# B&R Automation Studio project CombinedLinenCleanA6 (part 4)

#### usb_pmem.ab
```automation-basic
;--------------------------------------------------------------
;Copy BagData, C and D data to and from USB Mass Storage device
;--------------------------------------------------------------

;----------------------------------------------------
;Version 1.00 05/08/2006 D.J. First Issue
;Version 2.00 24/06/2009 D.J. Added D32 & VC_Posn
;Version 3.00 03/11/2010 D.J. Changed VC to RB (Robo)
;----------------------------------------------------

;Notes:-
;Add a mass storage device to the PLC CPU
;In CPU Properties select File Device
;Add a new device and set the Device Name to "USBStick"
;set the path of the USB device eg. "IF3.ST1" for a CP340

PROGRAM _INIT

bOK 			= FALSE
STEP 			= 1
byErrorLevel 	= 0
CurrentFile 	= 0

END_PROGRAM

PROGRAM _CYCLIC

;Error Step
IF STEP = 0 THEN
	bOK = FALSE
ENDIF

;Check if the file exists
IF STEP = 1 THEN

	FOpen.enable    = TRUE
    FOpen.pDevice   = "USBStick"
    IF CurrentFile = 0 THEN
    	FOpen.pFile     = "PLC_BagData.dat"
    ELSE IF CurrentFile = 1 THEN
    	FOpen.pFile     = "PLC_C.dat"
    ELSE IF CurrentFile = 2 THEN
    	FOpen.pFile     = "PLC_D.dat"
	ELSE IF CurrentFile = 3 THEN
    	FOpen.pFile     = "PLC_D32.dat"
	ELSE IF CurrentFile = 4 THEN
    	FOpen.pFile     = "PLC_RBPosn.dat"
    ENDIF
    FOpen.mode      = 2 ;Read and write access

    FOpen FUB FileOpen()

    dwIdent = FOpen.ident
    wStatus = FOpen.status

    ;Status - 20708 = File doesn't exist
    IF (wStatus = 20708) THEN
    	STEP = 2 ;If the file not found then create the file
    ELSE
    	IF (wStatus = 0) THEN
        	STEP = 4 ;If the file exists then copy back to PLC
    	ELSE
        	IF (wStatus <> 65535) THEN
            	byErrorLevel = 1
                STEP = 0
				IF (wStatus = 20799) THEN
                	wError = FileIoGetSysError()
           		ENDIF
            ENDIF
    	ENDIF
    ENDIF

ENDIF

;Create the file
IF STEP = 2 THEN

	FCreate.enable  = TRUE
    FCreate.pDevice = "USBStick"
    IF CurrentFile = 0 THEN
    	FCreate.pFile     = "PLC_BagData.dat"
    ELSE IF CurrentFile = 1 THEN
    	FCreate.pFile     = "PLC_C.dat"
    ELSE IF CurrentFile = 2 THEN
    	FCreate.pFile     = "PLC_D.dat"
    ELSE IF CurrentFile = 3 THEN
    	FCreate.pFile     = "PLC_D32.dat"
	ELSE IF CurrentFile = 4 THEN
    	FCreate.pFile     = "PLC_RBPosn.dat"
    ENDIF
    FCreate FUB FileCreate()

    dwIdent = FCreate.ident
    wStatus = FCreate.status

    IF (wStatus = 0) THEN
    	STEP = 3
    ELSE
    	IF (wStatus <> 65535) THEN
        	byErrorLevel = 4
            STEP = 5 ;Close
			IF (wStatus = 20799) THEN
            	wError = FileIoGetSysError() ;General System Error - get more info
        	ENDIF
    	ENDIF
    ENDIF
ENDIF

;Write data to the file
IF STEP = 3 THEN

    FWrite.enable   = TRUE
    FWrite.ident    = dwIdent
    FWrite.offset   = 0
    IF CurrentFile = 0 THEN
    	FWrite.pSrc     = pBag
    	FWrite.len      = sizeof(Bag)
    ELSE IF CurrentFile = 1 THEN
    	FWrite.pSrc     = pC
    	FWrite.len      = sizeof(C)
    ELSE IF CurrentFile = 2 THEN
    	FWrite.pSrc     = pD
    	FWrite.len      = sizeof(D)
	ELSE IF CurrentFile = 3 THEN
    	FWrite.pSrc     = pD32
    	FWrite.len      = sizeof(D32)
	ELSE IF CurrentFile = 4 THEN
    	FWrite.pSrc     = pRB_Posn
    	FWrite.len      = sizeof(RB_Posn)
    ENDIF

    FWrite FUB FileWrite()

    wStatus = FWrite.status

    ;Status
    IF (wStatus = 0) THEN
    	STEP = 5 ;Close
    ELSE
       	IF (wStatus <> 65535) THEN
        	byErrorLevel = 3
    		STEP = 0

          	IF (wStatus = 20799) THEN
            	wError = FileIoGetSysError() ;General System Error - get more info
        	ENDIF
     	ENDIF
  	ENDIF
ENDIF

;Read file
IF STEP = 4 THEN

    FRead.enable    = TRUE
    FRead.ident     = dwIdent
    FRead.offset    = 0

	IF CurrentFile = 0 THEN
    	FRead.pDest     = pBag
    	FRead.len      = sizeof(Bag)
    ELSE IF CurrentFile = 1 THEN
    	FRead.pDest     = pC
    	FRead.len      = sizeof(C)
    ELSE IF CurrentFile = 2 THEN
    	FRead.pDest     = pD
    	FRead.len      = sizeof(D)
    ELSE IF CurrentFile = 3 THEN
    	FRead.pDest     = pD32
    	FRead.len      	= sizeof(D32)
	ELSE IF CurrentFile = 4 THEN
    	FRead.pDest     = pRB_Posn
    	FRead.len      	= sizeof(RB_Posn)
	ENDIF

    FRead FUB FileRead()

    wStatus = FRead.status

	;Status
    IF (wStatus = 0) THEN
    	STEP = 5
    ELSE
        IF (wStatus <> 65535) THEN
            byErrorLevel = 4
            STEP = 0
            IF (wStatus = 20799) THEN
            	wError = FileIoGetSysError() ;General System Error - get more info
            ENDIF
        ENDIF
    ENDIF
ENDIF

;Close the file
IF STEP = 5 THEN

	FClose.enable   = TRUE
	FClose.ident    = dwIdent

	FClose FUB FileClose()

	wStatus = FClose.status

	;Status
	IF (wStatus = 0) THEN
		STEP = 7
	ELSE
        IF (wStatus <> 65535) THEN
            byErrorLevel = 5
            STEP = 0

            IF (wStatus = 20799) THEN
            	wError = FileIoGetSysError() ;General System Error - get more info
            ENDIF
        ENDIF
	ENDIF
ENDIF

;Operation Complete - try next file if required
IF STEP = 7 THEN
	IF CurrentFile < 4 THEN
		CurrentFile = CurrentFile + 1
		STEP = 1
	ENDIF
ENDIF

;Set this step manually to test this routine
IF (STEP = 8) THEN
	CurrentFile = 0
	STEP		= 1
ENDIF
END_PROGRAM
```

- Program Logical/Sequences/200ms/zzAlarms (IEC, version 4.00.0) (no source held here)

### zzstn_q.var
```iecst
VAR
	n : UINT;
	ValidWeight : BOOL;
	SP1Reached : BOOL;
	SP2Reached : BOOL;
	SP3Reached : BOOL;
	TestWeight : UINT;
	StnIntoQ : BOOL;
	StnsInQ : BOOL;
	PurgeStation : BOOL;
	StnsToPurge : BOOL;
	ManualRelease : BOOL;
	TestStation : UINT;
	z : UINT;
	Calibration : BOOL;
END_VAR
```

### Program Logical/Sequences/200ms/zzTime

#### zztime.var
```iecst
VAR RETAIN
	MiliSeconds	:UINT;
	Seconds	:UINT;
END_VAR

VAR
	TEST	:BOOL;
	TimeLast	:TIME;
	TimeNow	:TIME;
	TimeDiff	:TIME;
	SysRunning	:BOOL;
	ActionPLS	:BOOL;
	NoActionET	:TIME;
	NoAction	:BOOL;
	NoActionPLS	:BOOL;
	PLCFirstScan	:BOOL;
	Seq	:UINT;
	Minutes	:INT;
	Hours	:UINT;
	SysIdleMinutes	:UINT;
	SystemAction	:BOOL;
END_VAR
```

#### zztime.ab
```automation-basic
;-------------------
;System Running Time
;-------------------

;-----------------------------------------
;Revision 1.00 12/10/2005 D.J. First Issue
;-----------------------------------------

;Detection of system running - once the detection sequence has remained idle for a given
;period the clock is stopped and the idle time (minutes) is given back. If the idle time
;is 5 minutes and the system stopped at 12:01 then when the time is given back the time will
;read 12:-04 as the time is only taken from the minutes and no the hours count.

PROGRAM _INIT

PLCFirstScan = TRUE

END_PROGRAM

PROGRAM _CYCLIC

;Only use one sequence for system running. Norrmally Offgoing or a loop use the Discharger
D[905]	;Monitor

SystemAction = FALSE
IF D[915] <> Seq THEN
	SystemAction 	= TRUE
	Seq 			= D[915]
ENDIF

R_TRIG(SystemAction,ActionPLS)

TimeNow = clock_ms()

;System Start / Stop Running
IF ActionPLS THEN
	SysRunning 	= TRUE
ENDIF

SysIdleMinutes = 5

TON_10ms(NOT SystemAction,(SysIdleMinutes * 6000),NoAction,NoActionET)

;Read from Graphics
;Seconds = D[310]
Minutes = INT(D[311]) ;Can go minus
Hours	= D[312]

R_TRIG(NoAction,NoActionPLS)

;System has stopped give back the running timer time
IF NoActionPLS THEN
	Minutes 	= Minutes - SysIdleMinutes
	SysRunning 	= FALSE
ENDIF

IF TEST THEN
	Minutes 	= Minutes - 10
	TEST 		= FALSE
ENDIF

IF SysRunning THEN
	TimeDiff	= DiffT(TimeNow,TimeLast)
	MiliSeconds = MiliSeconds + UINT(TimeDiff)
ENDIF

TimeLast = TimeNow

;Count Seconds Running
IF MiliSeconds >= 1000 THEN
	Seconds 	= Seconds + 1
	MiliSeconds = MiliSeconds - 1000 ;Keep and remaing ms to be added next time
ENDIF

IF Seconds >= 60 THEN
	Minutes 	= Minutes + 1
	Seconds 	= Seconds - 60
ENDIF

IF Minutes >= 60 THEN
	Hours 		= Hours + 1
	Minutes	 	= Minutes - 60
ENDIF

;Count Each 1000 hours
IF Hours >= 1000 THEN
	D[313] 		= D[313] + 1
	Hours 		= Hours - 1000
ENDIF

;Store to Graphics
;D[310] = Seconds - don't display seconds as causes TCP/IP driver to send data to Graphics
D[311] = UINT(Minutes)
D[312] = Hours
D[313] = D[313] ;Hours * 1000

END_PROGRAM
```

### zzweigh.typ
```iecst
(********************************************************************
 * COPYRIGHT -- HP
 ********************************************************************
 * Package: NewPackage
 * File: zzweigh.typ
 * Author: treamsbottom
 * Created: April 10, 2014
 ********************************************************************
 * Data types of package NewPackage
 ********************************************************************)

TYPE
	enum_Calib :
		(
		Calib_Low,
		Calib_High
		);
END_TYPE
```

- Data object Logical/Sequences/Robo_Drive_Control/Param_0_25kwStar1 (Simple, version 4.00.0) (no source held here)

- Data object Logical/Sequences/Robo_Drive_Control/Param_2_2kwStar (Simple, version 4.00.0) (no source held here)

- Data object Logical/Sequences/Robo_Drive_Control/ParaTest (Simple) (no source held here)

- Program Logical/Sequences/TB/12_belt2 (IEC) (no source held here)

### zcusfifo.var
```iecst
VAR RETAIN
	OngoingCus	:UINT;
	EditCus	:UINT;
	n	:UINT;
	x	:UINT;
END_VAR
```

### Program Logical/Sequences/zzalarms (IEC, version 2.00.0)

#### zzalarms.var
```iecst
VAR RETAIN
	I_CancelAlarm	:BOOL;
END_VAR

VAR
	BuildD220	:UINT;
	AlmNumber	:UINT;
	n	:UINT;
	AlarmCount	:UINT;
	CancelBeacon	:BOOL;
	I_MotorOverload	:BOOL;
	UnloadingAlarm	:BOOL;
	I_InverterFault	:BOOL;
	BeaconInList	:BOOL;
END_VAR
```

#### zzalarmsCyclic.ab
```automation-basic
PROGRAM _CYCLIC
	(* cyclic program *)

;-----------------------------------------------
;Alarm Messages with Screen position and history
;-----------------------------------------------

;------------------------------------------------
;Version 1.00 - 08/12/2005 First Issue D.J.
;Vesrion 2.00 - 17/10/2006 Added Alarm.Extra D.J.
;------------------------------------------------

;Note - Sequence must set the following
;Alarm[x].on
;Alarm[x].Bag - for the bag position where the alarm will appear
;Alarm[x].Name - for the message that will be displayed use constants strating "alm"
;Alarn[x].Extra - Extra data for Graphics to use ie. Line number with fault on offgoing storage

I_CancelAlarm 	= FALSE ;X[4].X16
I_EStop 		= Std.EStop
I_MotorOverload = Std.MotorOverload
I_InverterFault = FALSE ;(X[3].X03 OR X[3].X04 OR X[3].X05 OR X[3].X06)

;--------------
;Alarm Messages
;--------------

IF I_EStop THEN
	Alarm[100].On	= TRUE
	Alarm[100].Bag 	= 0
	Alarm[100].Name	= almEmergencyStop
ELSE IF I_MotorOverload THEN
	Alarm[100].On	= TRUE
	Alarm[100].Bag 	= 0
	Alarm[100].Name	= almMotorOverload
ELSE IF I_InverterFault THEN
	Alarm[100].On	= TRUE
	Alarm[100].Bag 	= 0
	Alarm[100].Name	= almInverterFault
ELSE
	Alarm[100].On	= FALSE
	Alarm[100].Bag 	= 0
	Alarm[100].Name	= almNoAlarm
ENDIF

;Shuffle the Alarms List

AlarmCount 		= 0
BeaconInList 	= FALSE

LOOP n = 1 TO 10 DO

	;If Alarm not on anymore the clear from the list
	AlmNumber = D[200 + n]
	IF NOT Alarm[AlmNumber].On THEN
		D[200 + n] = 0
		D[210 + n] = 0
	ENDIF

	;Shuffle the list down
	IF (D[200 + n] = 0) AND (D[201 + n] > 0) AND (n <> 10) THEN
		D[200 + n] = D[201 + n]
		D[210 + n] = D[211 + n]
		D[201 + n] = 0
		D[211 + n] = 0
	ENDIF

	;Set InList for any alarm in the list
	Alarm[D[200 + n]].InList = TRUE

	;Calculate total alarms in the list
	IF D[200 + n] > 0 THEN
		AlarmCount = AlarmCount + 1
	ENDIF

	;Is the alarm beacon required?
	IF Alarm[AlmNumber].On AND Alarm[AlmNumber].Beacon THEN
		BeaconInList = TRUE
	ENDIF

ENDLOOP

;Cancel the alarm beacon
IF I_CancelAlarm THEN
	CancelBeacon = TRUE
ENDIF

;Cancel the CancelAlarm beacon if no alarm in the list requires the beacon
IF NOT BeaconInList THEN
	CancelBeacon = FALSE
ENDIF

;Look at each sequence alarm and if not in list then add to list if space
LOOP n = 1 TO 109 DO

	;If alarm active and a code has been given and not in the list and history is clear then add
	IF ((AlarmCount < 10) AND Alarm[n].On AND NOT Alarm[n].InList AND ((D[221] = 0) OR (n > 100))) THEN

		;If name not set then set to general
		IF (Alarm[n].Name = 0) THEN
			Alarm[n].Name = almGeneralSequence
		ENDIF

		D[210] 			= n
		BuildD220		= LSL(Alarm[n].Extra,8)
		BuildD220 		= BuildD220 + Alarm[n].Name
		D[220] 			= BuildD220

		;New alarm found requiring the beacon
		IF Alarm[n].Beacon THEN
			CancelBeacon = FALSE
		ENDIF

		;Store to History - if not Unloading Alarm
		IF (n <= 100) THEN
			D[221] 			= n				;Alarm Number (Seq)
			D[222]			= Alarm[n].Name	;Alarm Name / Message
			D[223] 			= D[223] + 1	;Alarm ID
			D[224]			= Alarm[n].Extra;Alarm Extra Data
			IF D[223] > 32000 THEN
				D[223] = 1
			ENDIF
		ENDIF

		;Inc Total Alarms
		AlarmCount = AlarmCount + 1

	ENDIF

	;Cancel All InList's - will be checked on the next scan
	Alarm[n].InList = FALSE

ENDLOOP

;Show Alarm position on the screen
IF D[201] > 0 THEN
	D[0] = Alarm[D[201]].Bag
ELSE
	D[0] = 0
ENDIF

UnloadingAlarm = Alarm[101].On OR Alarm[102].On OR Alarm[103].On OR Alarm[104].On

;Alarm Output - Unloading Alarm cannot be cancelled
Y[3].Y16 = ((BeaconInList AND NOT CancelBeacon) OR UnloadingAlarm)
;Y[4].Y15 = CancelAlarm
END_PROGRAM
```

### Program Logical/Sequences/zzbagsfl

#### zzbagsfl.var
```iecst
VAR RETAIN
	CurrentBag	:UINT;
	CurrentLine	:UINT;
	LineSp	:UINT;
END_VAR

VAR
	NextBag	:UINT;
END_VAR
```

#### zzbagsflCyclic.ab
```automation-basic
PROGRAM _CYCLIC
	(* cyclic program *)

;-----------------------------------------------------------
;Revision 1.00 19/12/2005 D.J. First Issue - Using BAG array
;-----------------------------------------------------------

Std.BagsWithDestinations 	= FALSE
Std.CustomerFound	 		= FALSE

IF (Bag[75].Cat>0)AND (Bag[5].Cat=0)THEN
		Bag[5] = Bag[75]
		Bag[75] = Bag[0]
ENDIF
IF (Bag[70].Cat>0)AND (Bag[20].Cat=0)THEN
		Bag[20] = Bag[70]
		Bag[70] = Bag[0]
ENDIF

LOOP CurrentLine = 1 to Std.MaxLinesBuffers DO

	LineSp = 0

	LOOP CurrentBag = Line[CurrentLine].FirstBag  TO Line[CurrentLine].LastBag DO

		EXITIF Line[CurrentLine].FirstBag = 0

		NextBag = (CurrentBag + 1)

		IF ((CurrentBag < Line[CurrentLine].LastBag) AND ((Bag[CurrentBag].Cat = 0) AND (Bag[NextBag].Cat > 0))) THEN

			;Copy Next Bag to Current
			Bag[CurrentBag]	= Bag[NextBag]
			Bag[NextBag] 	= Bag[0]

		ENDIF

		IF ((Bag[CurrentBag].Dst > 0) AND (CurrentLine <= Std.MaxLines)) THEN
			Std.BagsWithDestinations = TRUE
		ENDIF

		;Add the line spaces up
		IF Bag[CurrentBag].Cat = 0 THEN
			LineSp = (LineSp + 1)
		ENDIF

		;For Customer FIFO table
		;-----------------------
		;Customer at front of FIFO in Storage
		IF ((Bag[CurrentBag].Cus = D[401]) AND (D[401] > 0) AND (CurrentLine <= Std.MaxLines)) THEN
			Std.CustomerFound	 	= TRUE
		ENDIF

	ENDLOOP
	;Save the number of spaces on the current line
	Line[CurrentLine].Space = LineSp

ENDLOOP

Line[4].Space = (Line[4].Space + Line[10].Space)
Line[1].Space = (Line[1].Space + Line[11].Space)

END_PROGRAM
```

### Program Logical/Sequences/zzbitcal

#### zzbitcalCyclic.ab
```automation-basic
PROGRAM _CYCLIC
	(* cyclic program *)

	;-----------------------------------------------------------
	;Revision 1.00 19/12/2005 D.J. First Issue - Using BAG array
	;-----------------------------------------------------------

	;Find the Space on each Storage line including the Ongoing and Offgoing Bags In Transit

	;See Init Routine - Change settings for bags in transit bag numbers

	;Clear local calculation
	LOOP n = 1 TO Std.MaxLinesBuffers DO
		SpaceBIT[n] = 0
	ENDLOOP

	;Ensure the destination is less than the Array size of SpaceBIT	(normally 100)
	LOOP n = 1 TO TotalTransitBags DO
		Destination = Bag[BITDest[n]].Dst
		IF (Destination > 0) AND (Destination < 100) THEN
			SpaceBIT[Destination] = SpaceBIT[Destination] + 1
		ENDIF
	ENDLOOP

	;Once all calculated then update the global line space
	LOOP n = 1 TO Std.MaxLinesBuffers DO
		Spaces = (INT(Line[n].Space) - INT(SpaceBIT[n]))
		IF Spaces > 0 THEN
			Line[n].SpaceBIT = UINT(Spaces)
		ELSE
			Line[n].SpaceBIT = 0
		ENDIF
	ENDLOOP

END_PROGRAM
```

#### zzbitcalInit.ab
```automation-basic
PROGRAM _INIT
	(* init program *)

BITBag = 1

;Transfer Belt Bags - Pair loop
LOOP n = 32 TO 59 DO
	BITDest[BITBag] = n
	BITBag = BITBag + 1
ENDLOOP

;Bags in transit
;LOOP n = 140 to 179 DO
	;BITDest[BITBag] = n
	;BITBag = BITBag + 1
;ENDLOOP

TotalTransitBags = (BITBag - 1)
END_PROGRAM
```

- Program Logical/Sequences/zzclrmem (IEC, version 2.00.0) (no source held here)

### Program Logical/Sequences/zzconst (IEC, version 1.00.0)

#### zzconstInit.ab
```automation-basic
PROGRAM _INIT
	(* init program *)

Std.AutoMaticRelease   	= TRUE	;Set to TRUE for AutoMatic Release using setpoints. FALSE for Push-Button Release
Std.StationReports  	= TRUE  ;Transfer reports to PC

Std.PairingLoop   		= FALSE
Std.CustomerFIFO		= TRUE	;Use Customer FIFO Table

Std.MaxIO				= 39	;Max PLC I/O Cards - check X and Y array size

Std.MaxCats           	= 99	;Max Categories - Should be 99 or less Max = 255
Std.MaxCust           	= 999	;Max Customers
Std.MaxDischargers    	= 2		;Total Dischargers
Std.MaxLines          	= 11	    ;Max storage lines
Std.MaxLinesBuffers   	= 18	;Storage lines + Buffers
Std.MaxWeighstations  	= 16	    ;Total Weighstations
Std.MaxStationBanks		= 1		;Total Banks of sorting Stations
Std.MaxSearch			= 2    	;Include all station banks and Loading VC's etc
Std.StationBagsStart[1]	= 201	;Bag Number of first bank of sorting stations
Std.StationBagsStart[2] = 0 	;Bag Number of second bank of sorting stations
Std.MinReleaseWeight  	= 30	;Include 10ths Norm 30

Ldg[1].StartStn 		= 1 	;Bank 1 Start station number
Ldg[1].EndStn			= 16	    ;Bank 1 End station number

Ldg[2].StartStn 		= 0 	;Bank 2 Start station number
Ldg[2].EndStn			= 0		;Bank 2 End station number

;Enter the First and Last bag for all the Storage lines including buffers
Line[1].FirstBag = 1
Line[1].LastBag  = 5

Line[2].FirstBag = 6
Line[2].LastBag  = 10

Line[3].FirstBag = 11
Line[3].LastBag  = 13

Line[4].FirstBag = 16
Line[4].LastBag  = 20

Line[5].FirstBag = 26
Line[5].LastBag  = 29

Line[6].FirstBag = 21
Line[6].LastBag  = 24

Line[7].FirstBag = 63  ;New line for cdc7
Line[7].LastBag  = 66

Line[8].FirstBag = 78  ;New line for cdc8
Line[8].LastBag  = 81

Line[9].FirstBag = 0
Line[9].LastBag  = 0

Line[10].FirstBag = 70  ;Part of line 1
Line[10].LastBag  = 72

Line[11].FirstBag = 75  ;Part of line 4
Line[11].LastBag  = 77

Line[12].FirstBag = 0
Line[12].LastBag  = 0

Line[13].FirstBag = 0
Line[13].LastBag  = 0

Line[14].FirstBag = 0
Line[14].LastBag  = 0

Line[15].FirstBag = 0
Line[15].LastBag  = 0

Line[16].FirstBag = 51
Line[16].LastBag  = 52

Line[17].FirstBag = 38
Line[17].LastBag  = 38

Line[18].FirstBag = 53    ;New line for CP16
Line[18].LastBag  = 53

Line[19].FirstBag = 0
Line[19].LastBag  = 0

Line[20].FirstBag = 0
Line[20].LastBag  = 0

Line[21].FirstBag = 227
Line[21].LastBag  = 227

Line[22].FirstBag = 229
Line[22].LastBag  = 230

Line[23].FirstBag = 0
Line[23].LastBag  = 0

Line[24].FirstBag = 0
Line[24].LastBag  = 0

Line[25].FirstBag = 0
Line[25].LastBag  = 0

Line[26].FirstBag = 0
Line[26].LastBag  = 0

Line[27].FirstBag = 0
Line[27].LastBag  = 0

Line[28].FirstBag = 0
Line[28].LastBag  = 0

Line[29].FirstBag = 0
Line[29].LastBag  = 0

Line[30].FirstBag = 0
Line[30].LastBag  = 0

Line[31].FirstBag = 0
Line[31].LastBag  = 0

Line[32].FirstBag = 0
Line[32].LastBag  = 0

Line[33].FirstBag = 0
Line[33].LastBag  = 0

Line[34].FirstBag = 0
Line[34].LastBag  = 0
END_PROGRAM
```

#### zzconstCyclic.ab
```automation-basic
PROGRAM _CYCLIC
	(* cyclic program *)
;-----------------------------------------------------
;Revision A 01/05/2001 D.J. First Issue
;-----------------------------------------------------
;Code In Init Subroutine

Std.EnableOverUnderRelease = FALSE ;X6C 	;Override KeySwitch - See Stn_Q
END_PROGRAM
```

### Program Logical/Sequences/zzforcei

#### zzforcei.var
```iecst
VAR
	n	:UINT;
	XForce	:CardInputs;
	XForceVal	:CardInputs;
END_VAR
```

#### zzforceiCyclic.ab
```automation-basic
PROGRAM _CYCLIC
(* cyclic program *)

;---------------------------
;Input forcing from Graphics
;---------------------------

;Version 1.00 14/09/2006 D.J. First Issue

n = D[303]

IF (n > Std.MaxIO) THEN
	n = 0
ENDIF

XForce.X01 		= BIT_TST(D[304],0)
XForce.X02 		= BIT_TST(D[304],1)
XForce.X03 		= BIT_TST(D[304],2)
XForce.X04 		= BIT_TST(D[304],3)
XForce.X05 		= BIT_TST(D[304],4)
XForce.X06 		= BIT_TST(D[304],5)
XForce.X07 		= BIT_TST(D[304],6)
XForce.X08 		= BIT_TST(D[304],7)
XForce.X09 		= BIT_TST(D[304],8)
XForce.X10 		= BIT_TST(D[304],9)
XForce.X11 		= BIT_TST(D[304],10)
XForce.X12 		= BIT_TST(D[304],11)
XForce.X13 		= BIT_TST(D[304],12)
XForce.X14 		= BIT_TST(D[304],13)
XForce.X15 		= BIT_TST(D[304],14)
XForce.X16 		= BIT_TST(D[304],15)

XForceVal.X01 	= BIT_TST(D[305],0)
XForceVal.X02 	= BIT_TST(D[305],1)
XForceVal.X03 	= BIT_TST(D[305],2)
XForceVal.X04 	= BIT_TST(D[305],3)
XForceVal.X05 	= BIT_TST(D[305],4)
XForceVal.X06 	= BIT_TST(D[305],5)
XForceVal.X07 	= BIT_TST(D[305],6)
XForceVal.X08 	= BIT_TST(D[305],7)
XForceVal.X09 	= BIT_TST(D[305],8)
XForceVal.X10 	= BIT_TST(D[305],9)
XForceVal.X11 	= BIT_TST(D[305],10)
XForceVal.X12 	= BIT_TST(D[305],11)
XForceVal.X13 	= BIT_TST(D[305],12)
XForceVal.X14 	= BIT_TST(D[305],13)
XForceVal.X15 	= BIT_TST(D[305],14)
XForceVal.X16 	= BIT_TST(D[305],15)

X[n].X01 = (X[n].X01 AND NOT XForce.X01) OR (XForce.X01 AND XForceVal.X01)
X[n].X02 = (X[n].X02 AND NOT XForce.X02) OR (XForce.X02 AND XForceVal.X02)
X[n].X03 = (X[n].X03 AND NOT XForce.X03) OR (XForce.X03 AND XForceVal.X03)
X[n].X04 = (X[n].X04 AND NOT XForce.X04) OR (XForce.X04 AND XForceVal.X04)
X[n].X05 = (X[n].X05 AND NOT XForce.X05) OR (XForce.X05 AND XForceVal.X05)
X[n].X06 = (X[n].X06 AND NOT XForce.X06) OR (XForce.X06 AND XForceVal.X06)
X[n].X07 = (X[n].X07 AND NOT XForce.X07) OR (XForce.X07 AND XForceVal.X07)
X[n].X08 = (X[n].X08 AND NOT XForce.X08) OR (XForce.X08 AND XForceVal.X08)
X[n].X09 = (X[n].X09 AND NOT XForce.X09) OR (XForce.X09 AND XForceVal.X09)
X[n].X10 = (X[n].X10 AND NOT XForce.X10) OR (XForce.X10 AND XForceVal.X10)
X[n].X11 = (X[n].X11 AND NOT XForce.X11) OR (XForce.X11 AND XForceVal.X11)
X[n].X12 = (X[n].X12 AND NOT XForce.X12) OR (XForce.X12 AND XForceVal.X12)
X[n].X13 = (X[n].X13 AND NOT XForce.X13) OR (XForce.X13 AND XForceVal.X13)
X[n].X14 = (X[n].X14 AND NOT XForce.X14) OR (XForce.X14 AND XForceVal.X14)
X[n].X15 = (X[n].X15 AND NOT XForce.X15) OR (XForce.X15 AND XForceVal.X15)
X[n].X16 = (X[n].X16 AND NOT XForce.X16) OR (XForce.X16 AND XForceVal.X16)
END_PROGRAM
```

### Program Logical/Sequences/zzforceo

#### zzforceo.var
```iecst
VAR
	YForce	:CardOutputs;
	YForceVal	:CardOutputs;
	n	:UINT;
END_VAR
```

#### zzforceoCyclic.ab
```automation-basic
PROGRAM _CYCLIC
(* cyclic program *)

;----------------------------
;Output forcing from Graphics
;----------------------------

;Version 1.00 02/09/2006 D.J. First Issue

n = D[303]

IF (n > Std.MaxIO) THEN
	n = 0
ENDIF

YForce.Y01 		= BIT_TST(D[306],0)
YForce.Y02 		= BIT_TST(D[306],1)
YForce.Y03 		= BIT_TST(D[306],2)
YForce.Y04 		= BIT_TST(D[306],3)
YForce.Y05 		= BIT_TST(D[306],4)
YForce.Y06 		= BIT_TST(D[306],5)
YForce.Y07 		= BIT_TST(D[306],6)
YForce.Y08 		= BIT_TST(D[306],7)
YForce.Y09 		= BIT_TST(D[306],8)
YForce.Y10 		= BIT_TST(D[306],9)
YForce.Y11 		= BIT_TST(D[306],10)
YForce.Y12 		= BIT_TST(D[306],11)
YForce.Y13 		= BIT_TST(D[306],12)
YForce.Y14 		= BIT_TST(D[306],13)
YForce.Y15 		= BIT_TST(D[306],14)
YForce.Y16 		= BIT_TST(D[306],15)

YForceVal.Y01 	= BIT_TST(D[307],0)
YForceVal.Y02 	= BIT_TST(D[307],1)
YForceVal.Y03 	= BIT_TST(D[307],2)
YForceVal.Y04 	= BIT_TST(D[307],3)
YForceVal.Y05 	= BIT_TST(D[307],4)
YForceVal.Y06 	= BIT_TST(D[307],5)
YForceVal.Y07 	= BIT_TST(D[307],6)
YForceVal.Y08 	= BIT_TST(D[307],7)
YForceVal.Y09 	= BIT_TST(D[307],8)
YForceVal.Y10 	= BIT_TST(D[307],9)
YForceVal.Y11 	= BIT_TST(D[307],10)
YForceVal.Y12 	= BIT_TST(D[307],11)
YForceVal.Y13 	= BIT_TST(D[307],12)
YForceVal.Y14 	= BIT_TST(D[307],13)
YForceVal.Y15 	= BIT_TST(D[307],14)
YForceVal.Y16 	= BIT_TST(D[307],15)

Y[n].Y01 = (Y[n].Y01 AND NOT YForce.Y01) OR (YForce.Y01 AND YForceVal.Y01 AND NOT YForceDisable[n].Y01)
Y[n].Y02 = (Y[n].Y02 AND NOT YForce.Y02) OR (YForce.Y02 AND YForceVal.Y02 AND NOT YForceDisable[n].Y02)
Y[n].Y03 = (Y[n].Y03 AND NOT YForce.Y03) OR (YForce.Y03 AND YForceVal.Y03 AND NOT YForceDisable[n].Y03)
Y[n].Y04 = (Y[n].Y04 AND NOT YForce.Y04) OR (YForce.Y04 AND YForceVal.Y04 AND NOT YForceDisable[n].Y04)
Y[n].Y05 = (Y[n].Y05 AND NOT YForce.Y05) OR (YForce.Y05 AND YForceVal.Y05 AND NOT YForceDisable[n].Y05)
Y[n].Y06 = (Y[n].Y06 AND NOT YForce.Y06) OR (YForce.Y06 AND YForceVal.Y06 AND NOT YForceDisable[n].Y06)
Y[n].Y07 = (Y[n].Y07 AND NOT YForce.Y07) OR (YForce.Y07 AND YForceVal.Y07 AND NOT YForceDisable[n].Y07)
Y[n].Y08 = (Y[n].Y08 AND NOT YForce.Y08) OR (YForce.Y08 AND YForceVal.Y08 AND NOT YForceDisable[n].Y08)
Y[n].Y09 = (Y[n].Y09 AND NOT YForce.Y09) OR (YForce.Y09 AND YForceVal.Y09 AND NOT YForceDisable[n].Y09)
Y[n].Y10 = (Y[n].Y10 AND NOT YForce.Y10) OR (YForce.Y10 AND YForceVal.Y10 AND NOT YForceDisable[n].Y10)
Y[n].Y11 = (Y[n].Y11 AND NOT YForce.Y11) OR (YForce.Y11 AND YForceVal.Y11 AND NOT YForceDisable[n].Y11)
Y[n].Y12 = (Y[n].Y12 AND NOT YForce.Y12) OR (YForce.Y12 AND YForceVal.Y12 AND NOT YForceDisable[n].Y12)
Y[n].Y13 = (Y[n].Y13 AND NOT YForce.Y13) OR (YForce.Y13 AND YForceVal.Y13 AND NOT YForceDisable[n].Y13)
Y[n].Y14 = (Y[n].Y14 AND NOT YForce.Y14) OR (YForce.Y14 AND YForceVal.Y14 AND NOT YForceDisable[n].Y14)
Y[n].Y15 = (Y[n].Y15 AND NOT YForce.Y15) OR (YForce.Y15 AND YForceVal.Y15 AND NOT YForceDisable[n].Y15)
Y[n].Y16 = (Y[n].Y16 AND NOT YForce.Y16) OR (YForce.Y16 AND YForceVal.Y16 AND NOT YForceDisable[n].Y16)
END_PROGRAM
```

### Program Logical/Sequences/zzindi (IEC, version 1.00.0)

#### zzindi.var
```iecst
VAR
	n	:UINT;
	Encode	:ARRAY [0..4] OF BIT_ENCODE;
	Offset	:UINT;
END_VAR
```

### Program Logical/Sequences/zzio (IEC, version 3.00.0)

#### zzio.var
```iecst
VAR
	OutputCard	:BIT_ENCODE;
	CurrentCard	:UINT;
	InputCard	:BIT_ENCODE;
	n	:UINT;
END_VAR
```

#### zzioCyclic.ab
```automation-basic
PROGRAM _CYCLIC
(* cyclic program *)

;Transmit I/O to PC Graphics

;---------------------------------------------------------
;Version 1.00 19/12/2005 D.J. First Issue
;Version 2.00 13/11/2006 D.J. All I/O Sent to Graphics
;Version 3.00 02/05/2007 D.J. Do more than 1 card per scan
;---------------------------------------------------------

LOOP n = 1 TO 5 DO ;Do 5 cards per scan

	CurrentCard = CurrentCard + 1

	IF (CurrentCard > Std.MaxIO) THEN
		CurrentCard = 0
	ENDIF

	InputCard.Input[0] 	= X[CurrentCard].X01
	InputCard.Input[1] 	= X[CurrentCard].X02
	InputCard.Input[2] 	= X[CurrentCard].X03
	InputCard.Input[3] 	= X[CurrentCard].X04
	InputCard.Input[4] 	= X[CurrentCard].X05
	InputCard.Input[5] 	= X[CurrentCard].X06
	InputCard.Input[6] 	= X[CurrentCard].X07
	InputCard.Input[7] 	= X[CurrentCard].X08
	InputCard.Input[8] 	= X[CurrentCard].X09
	InputCard.Input[9] 	= X[CurrentCard].X10
	InputCard.Input[10] = X[CurrentCard].X11
	InputCard.Input[11] = X[CurrentCard].X12
	InputCard.Input[12] = X[CurrentCard].X13
	InputCard.Input[13] = X[CurrentCard].X14
	InputCard.Input[14] = X[CurrentCard].X15
	InputCard.Input[15] = X[CurrentCard].X16
	InputCard FUB BIT_ENCODE()

	D[500 + CurrentCard] 	= InputCard.Output

	OutputCard.Input[0] 	= Y[CurrentCard].Y01
	OutputCard.Input[1] 	= Y[CurrentCard].Y02
	OutputCard.Input[2] 	= Y[CurrentCard].Y03
	OutputCard.Input[3] 	= Y[CurrentCard].Y04
	OutputCard.Input[4] 	= Y[CurrentCard].Y05
	OutputCard.Input[5] 	= Y[CurrentCard].Y06
	OutputCard.Input[6] 	= Y[CurrentCard].Y07
	OutputCard.Input[7] 	= Y[CurrentCard].Y08
	OutputCard.Input[8] 	= Y[CurrentCard].Y09
	OutputCard.Input[9] 	= Y[CurrentCard].Y10
	OutputCard.Input[10] 	= Y[CurrentCard].Y11
	OutputCard.Input[11] 	= Y[CurrentCard].Y12
	OutputCard.Input[12] 	= Y[CurrentCard].Y13
	OutputCard.Input[13] 	= Y[CurrentCard].Y14
	OutputCard.Input[14] 	= Y[CurrentCard].Y15
	OutputCard.Input[15] 	= Y[CurrentCard].Y16
	OutputCard FUB BIT_ENCODE()

	D[600 + CurrentCard] 	= OutputCard.Output

ENDLOOP
END_PROGRAM
```

- Program Logical/Sequences/zzreport (IEC, version 1.00.0) (no source held here)

### Program Logical/Sequences/zzstatus

#### zzstatusCyclic.ab
```automation-basic
PROGRAM _CYCLIC
(* cyclic program *)

;System Status and Halting
;-------------------------

Std.StopSystem 				= (D[100] <> 0)

Std.EStop 					= NOT X[2].X15
Std.MotorOverload   		= X[2].X15 AND NOT X[2].X16
Std.SafetyOn				= X[2].X14
Std.HaltSys 				= NOT Std.SafetyOn ;OR Std.StopSystem)

;Indication[79]     	 		= Std.EStop ;EStop picture on graphics

;set to TRUE if not required
LoadingStopped 	= TRUE ;(Bag[220].Cat = 0)
OngoingStopped 	= TRUE ;(Bag[224].Cat = 0)
OffgoingStopped = TRUE ;(Bag[225].Cat = 0)

;If no Bag In Transit and stop requested then set system to stopped D[100] = 2
IF Std.StopSystem THEN
	IF LoadingStopped AND OngoingStopped AND OffgoingStopped THEN
		D[100] = 2
	ENDIF
ENDIF

;Force I/O Enable - Max ? Minutes
ForceEnable = X[8].X16

tmrForce.IN = ForceEnable
tmrForce.PT = 90000 ;6000 = 1 Minute
tmrForce FUB TON_10ms()

IF ForceEnable AND NOT tmrForce.Q THEN
	D[309] = 1
ELSE
	D[309] = 0
ENDIF

END_PROGRAM
```

- Program Logical/Sequences/zzstd (IEC, version 2.00.0) (no source held here)

### zzstn_q.var
```iecst
VAR RETAIN
	n	:UINT;
	ValidWeight	:BOOL;
	SP1Reached	:BOOL;
	SP2Reached	:BOOL;
	SP3Reached	:BOOL;
	TestWeight	:UINT;
	StnIntoQ	:BOOL;
	StnsInQ	:BOOL;
	PurgeStation	:BOOL;
	StnsToPurge	:BOOL;
END_VAR

VAR
	ManualRelease	:BOOL;
	TestStation	:UINT;
	z	:UINT;
END_VAR
```

### Program Logical/Sequences/zzstnmix

#### zzstnmix.var
```iecst
VAR
	n	:UINT;
	CatChanged	:BOOL;
	CatValid	:BOOL;
	CusChanged	:BOOL;
	CusValid	:BOOL;
	WgtValue	:INT;
	WgtValid	:BOOL;
	StnBag	:UINT;
END_VAR
```

#### zzstnmixCyclic.ab
```automation-basic
PROGRAM _CYCLIC
;----------------------
;Sorting Station Mixing
;----------------------

;----------------------------------------
;Version 1.00 09/12/2005 D.J. First Issue
;----------------------------------------

;Notes:
;When the operator changes either the Category or Customer of any station then the report should be written.
;If the Customer or Category is set to zero the report will be written for the previous Cat and Cus however
;the previous Cat and Cus will be set to zero. When the Cat or Cus is next changed there will be no report

IF Std.StationReports THEN

	;Special for Mewa only box 1 to 6 are reported on
	LOOP n = 1 TO Std.MaxWeighstations DO

		StnBag = n + (Std.StationBagsStart[1] - 1) ;Assumes all station bags will follow in order

		IF (ReportLoading[n].Cat = 0) THEN

			;Check if Category or Customer have been changed
			CatChanged 	= (Bag[StnBag].Cat <> StnPrev[n].Cat)
			CatValid   	= (StnPrev[n].Cat > 0)

			CusChanged 	= (Bag[StnBag].Cus <> StnPrev[n].Cus)
			CusValid   	= (StnPrev[n].Cus > 0)

			;Check if anything has been added and current weight is not less than the previous
			WgtValue 	= Stn[n].Weight	- INT(StnPrev[n].Wgt)
			WgtValid 	= (WgtValue > 0)

			;Ensure valid values as we report on either a weight or count change
			IF (WgtValue < 0) THEN
				WgtValue = 0
			ENDIF

			IF ((CatChanged OR CusChanged) AND CusValid AND CatValid AND WgtValid) THEN

				ReportLoading[n].Cat = StnPrev[n].Cat		;Category
				ReportLoading[n].Cus = StnPrev[n].Cus		;Customer
				ReportLoading[n].Wgt = UINT(WgtValue)		;Weight
				ReportLoading[n].Cnt = 0					;Count
				ReportLoading[n].Stn = n         			;Station
				ReportLoading[n].Mcn = 0					;Machine

			ENDIF

			;Set Previous to Current even if the Previous values were not valid
			IF (CatChanged OR CusChanged) THEN
				StnPrev[n].Cat = Bag[StnBag].Cat
				StnPrev[n].Cus = Bag[StnBag].Cus
				StnPrev[n].Wgt = Stn[n].Weight
				StnPrev[n].Cnt = 0
			ENDIF

		ENDIF

	ENDLOOP

ENDIF

END_PROGRAM
```

### Program Logical/Sequences/zztc2end (IEC, version 1.00.0)

#### zztc2endCyclic.ab
```automation-basic
PROGRAM _CYCLIC
(* cyclic program *)

TCScan[2].End = clock_ms()

TCScan[2].Time = UINT(TCScan[2].End - TCScan[2].Start)

IF (TCScan[2].Time < TCScan[2].Min) OR (TCScan[2].Min = 0) THEN
	TCScan[2].Min = TCScan[2].Time
ELSE IF TCScan[2].Time > TCScan[2].Max THEN
	TCScan[2].Max = TCScan[2].Time
	D[67] = TCScan[2].Max
ENDIF
END_PROGRAM
```

### Program Logical/Sequences/zztc2str

#### zztc2strCyclic.ab
```automation-basic
PROGRAM _CYCLIC
(* cyclic program *)

TCScan[2].Start = clock_ms()
END_PROGRAM
```

### Program Logical/Sequences/zztcpip (IEC, version 1.00.0)

#### zztcpipCyclic.ab
```automation-basic
PROGRAM _CYCLIC
;-----------------------------------
;TCP IP Driver Communications Driver
;-----------------------------------

;-----------------------------------------
;Revision 1.00 01/12/2005 D.J. First Issue
;-----------------------------------------

;Normally the driver will be sending constant requests - if the driver dosen't send anything for 1 second then the connection should be closed.

;------------
;Connection 1
;------------

;Restart - from init routine
IF ResetConnection THEN
	IF EnableConnection1 THEN
		NEWSTEP = 1
	ELSE
		NEWSTEP = 0
	ENDIF
ENDIF

STEP = NEWSTEP

;Disabled
IF STEP = 0 THEN
	;Do Nothing
ENDIF

;Init Server
IF STEP = 1 THEN
	TCPserv_1.enable = 1
	TCPserv_1.porta = 21001
	TCPserv_1 FUB TCPserv()
	IPAddr	= H_TO_NUDINT(TCPserv_1.ipaddr)
	Port	= TCPserv_1.portb
	NEWSTEP = 2
ENDIF

;Server to listening - until PC connects
IF STEP = 2 THEN
	TCPserv_1 FUB TCPserv()
	IPAddr	= H_TO_NUDINT(TCPserv_1.ipaddr)
	Port	= TCPserv_1.portb
	IF TCPserv_1.status = 0 THEN
		PLS = TRUE
		NEWSTEP = 3
	ELSE IF TCPserv_1.status = 27155 THEN 							;27155 = No buffer space available
		NEWSTEP = 6
	ENDIF
ENDIF

;PC Connected - if error then disconnect
IF STEP = 3 THEN

	WriteEnable = FALSE

	IF TCPsend_1.status = 0 THEN

		TCPrecv_1.enable = 1
		TCPrecv_1.cident = TCPserv_1.cident
		TCPrecv_1.buffer = ADR(rdata[0])
		TCPrecv_1.mxbuflng = SIZEOF(rdata)
		TCPrecv_1 FUB TCPrecv()
		RXLength = TCPrecv_1.rxbuflng
		RXStatus = TCPrecv_1.status

		IF RXLength > 0 THEN

			Data_RXTX_Type  = rdata[1] 								;WR = 1 BR = 2 WW = 3 BW = 4 - Bit Read and Bit Write not used
			Data_Array_Type = rdata[2]								;C  = 1 D  = 2 E  = 3 Bag = 4

			IF Data_Array_Type = 1 THEN
				Data_array_adr = pC
			ELSE IF Data_Array_Type = 2 THEN
				Data_array_adr = pD
			;ELSE IF Data_Array_Type = 3 THEN
			;	Data_array_adr = mem_adr_E
			ELSE IF Data_Array_Type = 3 THEN
				Data_array_adr = pBag
			ENDIF

			Data_StartH = rdata[3]
			Data_Start 	= LSL(Data_StartH,8) + rdata[4]
			Data_AmountH = rdata[5]
			Data_Amount = LSL(Data_AmountH,8) + rdata[6]

			PacketID = rdata[RXLength - 1] ;Packet ID sent back to Driver for check

			;Increase tx_frame size if limit changed  > 1000
			Data_Valid = ((Data_RXTX_Type > 0) AND (Data_Array_Type > 0) AND (Data_array_adr > 0) AND (Data_Amount > 0) AND (Data_Amount < 1001))

			LengthValid = (RXLength > (Data_Amount * 2))

			IF Data_Valid THEN

				RXValid = RXValid + 1

				IF (Data_RXTX_Type = 1) THEN					;Word Read - Transmit Data to PC

					tx_frame[0] = rdata[0]						;PLC Station

					memcpy(adr(tx_frame[1]),Data_array_adr + (Data_Start * 2),(Data_Amount * 2))

					tx_frame[(Data_Amount * 2) + 1] = PacketID ;USINT(0) ;Checksum not required
					tx_length 	= (Data_Amount * 2) + 2
					WriteEnable = TRUE

				ELSE IF (Data_RXTX_Type = 3) THEN 				;Word Write - Recieve data from PC

					memcpy(Data_array_adr + (Data_Start * 2),adr(rdata[7]),(Data_Amount * 2))

					tx_frame[0] = $06							;ACK
					tx_frame[1] = rdata[0]						;PLC Station
					tx_length 	= 2
					WriteEnable	= TRUE							;Set write enable

				ENDIF

			ELSE

				tx_frame[0] = $15 								;NAK
				tx_frame[1] = rdata[0] 							;PLC Station
				tx_length 	= 2
				WriteEnable	= TRUE								;Set write enable

			ENDIF

			IF WriteEnable THEN
				TCPsend_1.enable = 1
    			TCPsend_1.cident = TCPserv_1.cident
    			TCPsend_1.buffer = ADR(tx_frame[0])
    			TCPsend_1.buflng = tx_length ;SIZEOF(tx_frame)
    			TCPsend_1 FUB TCPsend()
	    	ENDIF

	    ENDIF

	ELSE
		TCPsend_1 FUB TCPsend()
	ENDIF

    IF (((TCPsend_1.status <> 0) AND (TCPsend_1.status <> 65535)) OR NoData) THEN
    	NoData  = FALSE
    	NEWSTEP = 4
    ENDIF

ENDIF
TON_10ms(((STEP = 3) AND (RXLength = 0)),500,NoData,NoDataET)

;Close the connection - if closed then go-to listen else go-to wait for close
IF STEP = 4 THEN
	TCPclose_1.enable = 1
	TCPclose_1.cident = TCPserv_1.cident
	TCPclose_1 FUB TCPclose()
	NEWSTEP = 5
ENDIF

;Closing - wait until connection closed
IF STEP = 5 THEN
	IF TCPclose_1.status <> 0 THEN
		TCPclose_1 FUB TCPclose()
	ELSE IF TCPclose_1.status = 0 THEN
		TCPsend_1.status = 0
		NEWSTEP = 1
	ENDIF
ENDIF

IF STEP = 6 THEN
	;Warm / Cold Start Required
ENDIF

;------------
;Connection 2
;------------

;Restart - from init routine
IF ResetConnection THEN
	IF EnableConnection2 THEN
		NEWSTEP2 = 1
	ELSE
		NEWSTEP2 = 0
	ENDIF
ENDIF

STEP2 = NEWSTEP2

;Disabled
IF STEP2 = 0 THEN
	;Do Nothing
ENDIF

;Init Server
IF STEP2 = 1 THEN
	TCPserv_2.enable = 1
	TCPserv_2.porta = 21002
	TCPserv_2 FUB TCPserv()
	IPAddr2	= H_TO_NUDINT(TCPserv_2.ipaddr)
	Port2	= TCPserv_2.portb
	NEWSTEP2 = 2
ENDIF

;Server to listening - until PC connects
IF STEP2 = 2 THEN
	TCPserv_2 FUB TCPserv()
	IPAddr2	= H_TO_NUDINT(TCPserv_2.ipaddr)
	Port2	= TCPserv_2.portb
	IF TCPserv_2.status = 0 THEN
		PLS2 = TRUE
		NEWSTEP2 = 3
	ELSE IF TCPserv_2.status = 27155 THEN								;27155 = No buffer space available
		NEWSTEP2 = 6
	ENDIF
ENDIF

;PC Connected - if error then disconnect
IF STEP2 = 3 THEN

	WriteEnable2 = FALSE

	IF TCPsend_2.status = 0 THEN

		TCPrecv_2.enable = 1
		TCPrecv_2.cident = TCPserv_2.cident
		TCPrecv_2.buffer = ADR(rdata2[0])
		TCPrecv_2.mxbuflng = SIZEOF(rdata2)
		TCPrecv_2 FUB TCPrecv()
		RXLength2 = TCPrecv_2.rxbuflng
		RXStatus2 = TCPrecv_2.status

		IF RXLength2 > 0 THEN

			Data_RXTX_Type  = rdata2[1] 								;WR = 1 BR = 2 WW = 3 BW = 4 - Bit Read and Bit Write not used
			Data_Array_Type = rdata2[2]									;C  = 1 D  = 2 E  = 3

			IF Data_Array_Type = 1 THEN
				Data_array_adr = pC
			ELSE IF Data_Array_Type = 2 THEN
				Data_array_adr = pD
			;ELSE IF Data_Array_Type = 3 THEN
			;	Data_array_adr = mem_adr_E
			ELSE IF Data_Array_Type = 3 THEN
				Data_array_adr = pBag
			ENDIF

			Data_StartH = rdata2[3]
			Data_Start 	= LSL(Data_StartH,8) + rdata2[4]
			Data_AmountH = rdata2[5]
			Data_Amount = LSL(Data_AmountH,8) + rdata2[6]

			PacketID = rdata2[RXLength2 - 1] ;Packet ID sent back to Driver for check

			Data_Valid = ((Data_RXTX_Type > 0) AND (Data_Array_Type > 0) AND (Data_array_adr > 0) AND (Data_Amount > 0) AND (Data_Amount < 1001))

			LengthValid = (RXLength2 > (Data_Amount * 2))

			IF Data_Valid THEN

				RXValid2 = RXValid2 + 1

				IF (Data_RXTX_Type = 1) THEN							;Word Read - Transmit Data to PC

					tx_frame2[0] = rdata2[0] 							;PLC Station

					memcpy(adr(tx_frame2[1]),Data_array_adr + (Data_Start * 2),(Data_Amount * 2))

					tx_frame2[(Data_Amount * 2) + 1] = PacketID ;USINT(0) ;Checksum not required
					tx_length2 	= (Data_Amount * 2) + 2
					WriteEnable2 = TRUE

				ELSE IF (Data_RXTX_Type = 3) THEN 						;Word Write - Recieve data from PC

					memcpy(Data_array_adr + (Data_Start * 2),adr(rdata2[7]),(Data_Amount * 2))

					tx_frame2[0] = $06									;ACK
					tx_frame2[1] = rdata2[0] 							;PLC Station
					tx_length2 	= 2
					WriteEnable2	= TRUE								;Set write enable

				ENDIF

			ELSE

				tx_frame2[0] = $15 										;NAK
				tx_frame2[1] = rdata2[0] 								;PLC Station
				tx_length2 	 = 2
				WriteEnable2 = TRUE										;Set write enable

			ENDIF

			IF WriteEnable2 THEN
				TCPsend_2.enable = 1
    			TCPsend_2.cident = TCPserv_2.cident
    			TCPsend_2.buffer = ADR(tx_frame2[0])
    			TCPsend_2.buflng = tx_length2 ;SIZEOF(tx_frame)
    			TCPsend_2 FUB TCPsend()
	    	ENDIF

	    ENDIF

	ELSE
		TCPsend_2 FUB TCPsend()
	ENDIF

    IF (((TCPsend_2.status <> 0) AND (TCPsend_2.status <> 65535)) OR NoData2) THEN
    	NoData2  = FALSE
    	NEWSTEP2 = 4
    ENDIF

ENDIF
TON_10ms(((STEP2 = 3) AND (RXLength2 = 0)),500,NoData2,NoData2ET)

;Close the connection - if closed then go-to listen else go-to wait for close
IF STEP2 = 4 THEN
	TCPclose_2.enable = 1
	TCPclose_2.cident = TCPserv_2.cident
	TCPclose_2 FUB TCPclose()
	NEWSTEP2 = 5
ENDIF

;Closing - wait until connection closed
IF STEP2 = 5 THEN
	IF TCPclose_2.status <> 0 THEN
		TCPclose_2 FUB TCPclose()
	ELSE IF TCPclose_2.status = 0 THEN
		TCPsend_2.status = 0
		NEWSTEP2 = 1
	ENDIF
ENDIF

IF STEP2 = 6 THEN
	;Warm / Cold Start Required
ENDIF

;Clear Reset Connection from Init Sub
ResetConnection = FALSE
END_PROGRAM
```

### Program Logical/Sequences/zztrip (IEC, version 1.00.0)

#### zztripCyclic.ab
```automation-basic
PROGRAM _CYCLIC
(* cyclic program *)

;--------------------------------------------------------------------------
;Primary trolley counting trips - ensure the main program can see the input
;--------------------------------------------------------------------------

CountTrip[1]  = X[6].X06 ;Bag on line 1
CountTrip[2]  = X[3].X05 ;            2
CountTrip[3]  = X[6].X07 ;            3
CountTrip[4]  = X[6].X05 ;            4
CountTrip[5]  = X[5].X15 ;Bag out sdc1
CountTrip[6]  = X[5].X11 ;            6
CountTrip[7]  = X[5].X16 ;            7
CountTrip[8]  = X[7].X12 ;            8
CountTrip[9]  = X[6].X10 ;            9
CountTrip[10] = X[4].X10 ;           10
CountTrip[11] = X[7].X11 ;           11
CountTrip[12] = X[7].X06 ;           12
CountTrip[13] = X[7].X08 ;           13
CountTrip[14] = X[4].X06 ;           14
CountTrip[15] = X[8].X04
CountTrip[16] = X[5].X01 ;SVC1 Buffer full
CountTrip[17] = X[5].X09 ;Bag on buffer line A
CountTrip[18] = X[2].X11 ;Bag out of svc2
;CountTrip[19] = X[7].X03 ;Sdc4 Bag Out
;CountTrip[20] = X[6].X12 ;Sdc3 Bag Out
;CountTrip[21] = X[6].X16 ;Sdc1 buffer line full
;CountTrip[22] = X[6].X15 ;Sdc2 buffer line full
;CountTrip[23] = X[9].X16 ;Sdc3 buffer line full
;CountTrip[24] = X[9].X14 ;Sdc4 buffer line full
;CountTrip[25] = X[9].X12 ;Sdc5 buffer line full
;CountTrip[26] = X[7].X07 ;Sdc5 Bag Out
;CountTrip[27] = X[6].X05 ;Bag out of sdc1
;CountTrip[28] = X[6].X08 ;Bag out of sdc2
;CountTrip[29] = X[7].X08 ;Sbc1 Buffer line full
;CountTrip[30] = X[3].X11 ;Sic1 buffer line full
;CountTrip[31] = X[7].X13 ;Bag out of svc3
;CountTrip[32] = X[10].X06 ;Bag out offgoing bag stacker
;CountTrip[33] = X[8].X06 ; Bag out of loading unit
;CountTrip[34] = X[4].X16
;CountTrip[35] = X[7].X16 ;Sbc1 Bag out
;CountTrip[36] = X[3].X12 ;Bag on transit line B

LOOP n = 1 TO 22 DO

	TripPLS[n].CLK = CountTrip[n]
	TripPLS[n] FUB R_TRIG()

	IF TripPLS[n].Q AND Timer[n].Q AND (C[n] < 2) THEN
		C[n] = C[n] + 1
	ENDIF

	Timer[n].IN = NOT CountTrip[n]
	Timer[n].PT = 10 ;100 = 1second
	Timer[n] FUB TON_10ms()

	Line[n].Full 	= (C[n] = 1)
	Line[n].Clear 	= ((C[n] >= 2) AND Timer[n].Q)

	Line[n].Trip	= (((CountOld[n] <> C[n]) AND (C[n] <> 0)) OR CountTrip[n]) ;Use for Bag Arrived at destination
	CountOld[n] 	= C[n]

ENDLOOP
END_PROGRAM
```

### Program Logical/Sequences/zzuld_3

#### zzuld_3.var
```iecst
VAR RETAIN
	TestDischarger	:UINT;
	BufferLineNum	:ARRAY [0..19] OF UINT;
	SearchSpaces	:UINT;
	BagsRemaining	:UINT;
	StepsSearched	:UINT;
	PriorityLine	:UINT;
	Quantity	:UINT;
	ManualBags	:UINT;
	CurrentBag	:UINT;
	FindBest	:UINT;
	RecircSpaces	:UINT;
	ExpressBag	:UINT;
	CatValid	:BOOL;
	RecircSpacesRemain	:UINT;
	SpacesUsed	:UINT;
	LastDischarger	:UINT;
	DepthValid2	:BOOL;
	PLS	:BOOL;
	Discharger	:UINT;
	FoundBag	:ARRAY [0..4] OF UINT;
	ExpressLine	:UINT;
	n	:UINT;
	LineDepthAllowed	:ARRAY [0..49] OF USINT;
	DepthValid	:BOOL;
	BatchSize	:UINT;
	LineValid	:BOOL;
	RegOffset	:ARRAY [0..19] OF UINT;
	RecirculationMaxDepth	:UINT;
	EndDischarger	:UINT;
	StartDischarger	:UINT;
	MatchCat2Cus1	:BOOL;
	ProgQtyComplete	:UINT;
	DischargerSpaces	:UINT;
	MatchCat3Cus1	:BOOL;
	ManualLine	:UINT;
	DischargerReady	:BOOL;
	ProgramFinished	:BOOL;
	NoBagAvailable	:BOOL;
	CustomerMode	:UINT;
	MatchCat1Cus1	:BOOL;
	MixCategories	:BOOL;
	LinesSearched	:UINT;
	MixCustomers	:BOOL;
	SearchCus	:ARRAY [0..3] OF UINT;
	ScanCount	:UINT;
	SearchCat	:ARRAY [0..3] OF UINT;
	SearchLine	:UINT;
	CurrentLine	:UINT;
	Dest	:UINT;
	CurrentDepth	:UINT;
	StartLine	:UINT;
	SkipIncompleteStep	:BOOL;
	AutoRepeat	:BOOL;
	ProgramReset	:BOOL;
	x	:UINT;
	CusValid	:BOOL;
	UnusedStep	:BOOL;
	ManualLineRecirc	:UINT;
	ManualBagsRecirc	:UINT;
	EndLineSearch	:UINT;
	StartLineSearch	:UINT;
	UldStep	:UINT;
	ProgramStep	:UINT;
	ProgramRunning	:BOOL;
	FoundLine	:UINT;
END_VAR

VAR
	AutoRecirculation	:BOOL;
	UnloadingMaxDepth	:UINT;
END_VAR
```

#### zzuld_3Init.ab
```automation-basic
PROGRAM _INIT
	;init program
	;------------

	;Constants
	;---------

	UnloadingMaxDepth 	= 7 ;Set with Batch Size and Scan Time in mind 8 = Standard

	StartDischarger 	= 1
	EndDischarger   	= 2

	StartLineSearch 	= 1
	EndLineSearch 		= 11

	RegOffset[1]    	= 1000
	RegOffset[2]    	= 1200
	RegOffset[3]    	= 1400
	RegOffset[4]    	= 1600
	RegOffset[5]    	= 1800

	;Enter Line Number for Discharger buffers - Recirc is after last Discharger
	;Destination Code bag will be allocated
	BufferLineNum[1]	= 12
	BufferLineNum[2]	= 13
	;BufferLineNum[3]	= 23
	;BufferLineNum[4]	= 24

	PriorityLine	= 0		;Always Search this line first then use the Uld[n].DischargerStartLine Set to 0 if not required
END_PROGRAM
```

- Library Logical/Libraries/SupLib4 (IEC, version 1.00.0) - Supertrack Systems Functions 4 (no source held here)

### Library Logical/Libraries/WETCAN2 (IEC, version 3.06.2)
Depends on: AsString, AsTime, CAN_LIB, DataObj, brsystem, runtime

#### WETCAN2.var
```iecst
VAR CONSTANT
	WC2_COMM_DIRECTION_READ	:USINT	:=0;
	WC2_COMM_DIRECTION_WRITE	:USINT	:=1;
	WC2_MODE_RW_CYCLIC	:INT	:=0;
	WC2_MODE_RW_EVENTCONTROLLED	:INT	:=1;
END_VAR
```

#### _GetNumberOfCan1Tels.ab
```automation-basic
FUNCTION_BLOCK _GetNumberOfCan1Tels
;********************************************************************************************************
; * Implementation of _GetNumberOfCan1Tels
;********************************************************************************************************
; * version 		3.6.1
; * last change		160112
; * by				H.O.
;********************************************************************************************************
; History:
; V3.6.1 - ###HO - 160112
;	* 306 # 3->2
;	* 316 # 2->1
;	* 361 # 3->2
;	* 371 # 2->1
; V3.6.0 - ###HO - 120210
;	* COB120 auch für ID 150,160,170,180,190
;	* COB121 auch für ID 151,161,171,181,191
; * V3.4.0 ###HO 211209
;	* COB ID 110 + 111
; V3.2.1 - ###hcs/HO - 111007
; 	COB_ID130und140 und COB_ID131und141 entfernt - stattdessen Neudefinition:
; 		* COB 130 und COB140 wie COB120
;		* COB131 und COB141 wie COB121
; * V3.2.0 ###HO 040907
;	* COBs 261+262 neu
;  	* COBs 302,303,304 wie 301 - 312,313,314 wie 311 - 253,255 wie 251 - 254,256 wie 252 - 352,353,354 wie 351
; * V 1.0.0 HO
; * V 2.0.0 HO
;	* COBs  123,251,252,480,481 added
; 	* COB 122 number of tels changed from two to four
; * V2.1.0	HO	070404
; 	* COB441..459 hinzugefügt
; * V2.1.5	HO	310805
; 	* COB401..419 hinzugefügt
; * V3.0.0	HO	010905
; 	* COBxxx.Customize[0..6] hinzugefügt -> Anzahl Telegramme inkrementiert
;	*  ###HO - 070905 neu ab V3.0.0
; 		*COBs 251=253=255=257 + 252=254=256=258
;	* COBs 307+317 hinzugefügt
; * V3.0.7 COB254,256,258:: 2->3
; * V3.1.0 COB126,127,128,129 hinzugefügt
;********************************************************************************************************

; this FUB returns the number of CAN1 telegrams
; - the CAN2 telegram will be divided up in this number of CAN1 telegrams later
; note: number of CAN1 telegrams depends on control byte's data of CAN2 structure !
; the number of telegrams is defined in CAN2 standard.

; 	-> 	pPV						..incoming pointer to PV to get info how many CAN1 telegrams should be broadcasted
;	-> 	ObjNr					..position of control byte's data depends on individual ID
; 		iNumberOfCan1Tels ->	..return value (see above)
;********************************************************************************************************
;********************************************************************************************************
; supported CANIDs: 120,121,122,123,130,140,131,141,201,209,211,219,221,231,
; 					301,306,311,316,351,361..369,371..379,401..419,421..439,441..459
; ###HO - 070905 neu ab V3.0.0
; COBs 251..256
;********************************************************************************************************

; !! be aware: UDINTs on intel targets start at addresses dividable by four !!
TARGETInfo_1.enable		= 1
TARGETInfo_1.pOSVersion	= adr(szOsVersion)
TARGETInfo_1 FUB TARGETInfo()

; get pointer to PV to identify AKZ..
memcpy(adr(LocalPV),pPV,sizeof(LocalPV))

iStatus = 0

case uiObjNr of
	action 110:
		iNumberOfCan1Tels = 3
	endaction
	action 111:
		iNumberOfCan1Tels = 2
	endaction
	action 120:
	action 126:
	action 128:
	action 130:
	action 140:
	action 150:
	action 160:
	action 170:
	action 180:
	action 190:
		; write AKZ to temporarily byte..
		byteTemp = LocalPV[13]
		if ( byteTemp = 1 ) then 	; AKZ has to be transmitted by tel three and four..
			iNumberOfCan1Tels = 5
		else 						; without AKZ -> broadcast only two telegrams..
			iNumberOfCan1Tels = 3
		endif
	endaction
	action 121:
	action 127:
	action 129:
	action 131:
	action 141:
	action 151:
	action 161:
	action 171:
	action 181:
	action 191:
		; for 121 only one tel defined
		iNumberOfCan1Tels = 2
	endaction
	action 122:
		; for 122 only two tels defined
		iNumberOfCan1Tels = 5
	endaction ; 122

	action 123:
		; for 123 only one tel defined
		iNumberOfCan1Tels = 2
	endaction ; 123
(*
	action 1130: ; 08.10.2007 - (hcs) DEAKTIVIERT
		if (TARGETInfo_1.DataFormat = 1) then ; intel
			; write AKZ to temporarily byte..
			byteTemp = LocalPV[17]
			if ( byteTemp = 1 ) then 	; AKZ has to be transmitted by tel three and four..
				iNumberOfCan1Tels = 5
			else 						; without AKZ -> broadcast only two telegrams..
				iNumberOfCan1Tels = 3
			endif
		else if (TARGETInfo_1.DataFormat = 2) then  ; motorola
			; write AKZ to temporarily byte..
			byteTemp = LocalPV[15]
			if ( byteTemp = 1 ) then 	; AKZ has to be transmitted by tel three and four..
				iNumberOfCan1Tels = 5
			else 						; without AKZ -> broadcast only two telegrams..
				iNumberOfCan1Tels = 3
			endif
		else
			iStatus = TARGETInfo_1.status
		endif
	endaction ; 130

	action 1131:	; 08.10.2007 - (hcs) DEAKTIVIERT
		iNumberOfCan1Tels = 2
	endaction ; 131

	action 140:
		if (TARGETInfo_1.DataFormat = 1) then ; intel
			; write AKZ to temporarily byte..
			byteTemp = LocalPV[17]
			if ( byteTemp = 1 ) then 	; AKZ has to be transmitted by tel three and four..
				iNumberOfCan1Tels = 5
			else 						; without AKZ -> broadcast only two telegrams..
				iNumberOfCan1Tels = 3
			endif
		else if (TARGETInfo_1.DataFormat = 2) then  ; motorola
			; write AKZ to temporarily byte..
			byteTemp = LocalPV[15]
			if ( byteTemp = 1 ) then 	; AKZ has to be transmitted by tel three and four..
				iNumberOfCan1Tels = 5
			else 						; without AKZ -> broadcast only two telegrams..
				iNumberOfCan1Tels = 3
			endif
		else
			iStatus = TARGETInfo_1.status
		endif
	endaction ; 140

	action 141:
		iNumberOfCan1Tels = 2
	endaction
*)
	action 201:
		iNumberOfCan1Tels = 3
	endaction
	action 209:
		iNumberOfCan1Tels = 3
	endaction
	action 211:
		iNumberOfCan1Tels = 2
	endaction
	action 219:
		iNumberOfCan1Tels = 2
	endaction
	action 221:
		iNumberOfCan1Tels = 3
	endaction
	action 231:
		iNumberOfCan1Tels = 2
	endaction
	action 251:
	action 253:
	action 255:
	action 257:
		iNumberOfCan1Tels = 3
	endaction

	action 252:
	action 254:
	action 256:
	action 258:
		iNumberOfCan1Tels = 2
	endaction

	action 261:
		iNumberOfCan1Tels = 1
	endaction
	action 262:
		iNumberOfCan1Tels = 1
	endaction
	action 301:
	action 302:
	action 303:
	action 304:
		iNumberOfCan1Tels = 3
	endaction

	action 306:
		iNumberOfCan1Tels = 3
	endaction
	action 307:
		iNumberOfCan1Tels = 3
	endaction
	action 311:
	action 312:
	action 313:
	action 314:
		iNumberOfCan1Tels = 2
	endaction

	action 316:
		iNumberOfCan1Tels = 2
	endaction
	action 317:
		iNumberOfCan1Tels = 2
	endaction
	action 351:
	action 352:
	action 353:
	action 354:
		iNumberOfCan1Tels = 3
	endaction
	action 361..369:
		iNumberOfCan1Tels = 3
	endaction
	action 371..379:
		iNumberOfCan1Tels = 2
	endaction
	action 401..419:
		iNumberOfCan1Tels = 3
	endaction
	action 421..439:
		; always four for this uiObjNr..
		iNumberOfCan1Tels = 4
	endaction
	action 441..459:
		iNumberOfCan1Tels = 2
	endaction
	action 480:
		iNumberOfCan1Tels = 3
	endaction
	action 481:
		iNumberOfCan1Tels = 3
	endaction

	; return error status 110 -> unsupported uiObjNr/uiCANID has been passed..
	elseaction:
		iStatus = 110;
	endaction
endcase

;********************************************************************************************************
;********************************************************************************************************
END_FUNCTION_BLOCK
```
